# EPICS StreamDevice protocol: oerconeSup/oercone.proto
Terminator = CR LF;

# How Oerlikon Centre-One Pressure Gauge Works:
## Send a command, then wait 100ms and send an ENQ (05 in Hex) to get the reply

getPressure {
	out "PR1";
	wait 100;
    in ACK;
	out ENQ;
	in "%d,%f";
}

getUnits {
    out "UNI";
	wait 100;
    in ACK;
	out ENQ;
    in "%{0|1|2|3}";
}

setUnits {
    #UNI,1 = mbar
    #UNI,2 = Torr
    #UNI,3 = Pascal
	#UNI,4 = Micron
    out "UNI,%{0|1|2|3}";
    in ACK;
}
